# EPICS autosave request: norhofLN2/norhofLN2_settings.req
$(P):DISABLE
